(* IEC 61131-3 sources: plc_on_fpga_riscv_hybrid/RV_FPGA_PLC_IDE_Projects/Timer_Test_4_1, 1 file *)

(* ---- Timer_Test_4_1.il ---- *)
VAR
    TON_1   : TON
    E_T   : TIME
END_VAR

PROGRAM Timer_Test_4_1
    R1 :
        CAL TON_1(
            IN := %SW.0,
            PT := T#1s,
            ET => E_T,
            Q  => %LEDG.0)
    R2 :
        LD     E_T
        TIME_TO_BOOL
        ST     %LEDR.0
END_PROGRAM
